// TIA Portal V16 export
// export: Created 2021-04-06T19:52:13.8560566Z, ExportSetting WithDefaults, DisplayName Totally Integrated Automation Portal, DisplayVersion V16, DisplayName TIA Portal Version Control Interface, DisplayVersion V16, DisplayName TIA Portal Openness, DisplayVersion V16, DisplayName STEP 7 Professional, DisplayVersion V16, DisplayName STEP 7 Safety, DisplayVersion V16, DisplayName WinCC Unified SCADA Engineering System, DisplayVersion V16
FUNCTION_BLOCK "ManualMode"   // FB10, LAD
{ S7_Optimized_Access := 'TRUE' }
VERSION : 0.1
// stored: AutoNumber false, IsIECCheckEnabled false, IsRetainMemResEnabled false, MemoryReserve 100, SetENOAutomatically false, UDAEnableTagReadback false
   VAR
      Bunker_Left : Array[0..12] of "controlValve";
      Bunker_Right { S7_SetPoint := 'True'} : Array[0..12] of "controlValve";
      Door { S7_SetPoint := 'True'} : Array[0..12] of "controlValve";
      flipper : "controlValve";
      runAll : Struct
         vibroLot : Bool;
      END_STRUCT;
      stopAlarm { S7_SetPoint := 'True'} : Bool;   // Стоп для блоков управления задвижками
   END_VAR
   VAR_TEMP
      i : Int;
   END_VAR
BEGIN

REGION Network 1: формирование AlarmStop
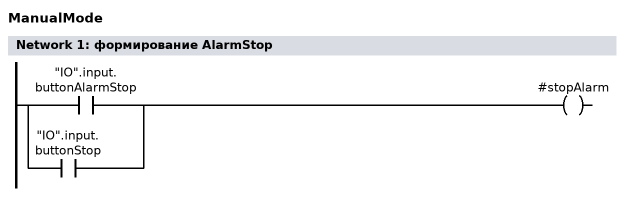
   RUNG wire#powerrail
      Contact( "IO".input.buttonAlarmStop )
      wire#w1
      Coil( #stopAlarm )
   END_RUNG
   RUNG wire#powerrail
      Contact( "IO".input.buttonStop )
   END_RUNG wire#w1
   // the same network as SCL:
   #stopAlarm := "IO".input.buttonAlarmStop OR "IO".input.buttonStop;
END_REGION

REGION Network 2 (SCL): ручное управление
   #i := 0;
   FOR #i := 1 TO 12 DO
       //если имеется разрешение на включение механизмов в ручном режиме
       IF "signalKVSStation".enableManualMode THEN
           //Bunker_left
           #Bunker_Left[#i](openQ => "signalKVSStation".qManualMode.Bunker_leftOpen[#i],
                            closeQ => "signalKVSStation".qManualMode.Bunker_leftClose[#i],
                            open := "hmi".weightLine[#i].manOpenLeftValveWeightPocket,
                            close := "hmi".weightLine[#i].manCloseLeftValveWeightPocket,
                            "time_open/close" := t#250ms,
                            stopAlarm := #stopAlarm);


           //Bunker_right
           #Bunker_Right[#i](openQ => "signalKVSStation".qManualMode.Bunker_rightOpen[#i],
                             closeQ => "signalKVSStation".qManualMode.Bunker_rightClose[#i],
                             open := "hmi".weightLine[#i].manOpenRightValveWeightPocket,
                             close := "hmi".weightLine[#i].manCloseRightValveWieghtPocket,
                             "time_open/close" := t#250ms,
                             stopAlarm := #stopAlarm);

           //Door
           #Door[#i](openQ => "signalKVSStation".qManualMode.Door_open[#i],
                     closeQ => "signalKVSStation".qManualMode.Door_close[#i],
                     open := "hmi".weightLine[#i].manOpenValveAfterVibroLot,
                     close := "hmi".weightLine[#i].manCloseValveAfterVibroLot,
                     "time_open/close" := t#250ms,
                     stopAlarm := #stopAlarm);

           //vibroLot
           IF "hmi".weightLine[#i].manVibroLotStart THEN
               "signalKVSStation".qManualMode.vibroLot[#i] := true;
           ELSE
               "signalKVSStation".qManualMode.vibroLot[#i] := false;
           END_IF;

           //теперь все что на два цикла
           IF #i = 1 OR #i = 2 THEN

               //Conv_FRV //Conv_REV
               IF "hmi".outConvAndPack[#i].manStartOutConv THEN
                   IF "hmi".outConvAndPack[#i].manIsUpConv THEN
                       "signalKVSStation".qManualMode.Conv_FRV[#i] := true;
                       "signalKVSStation".qManualMode.Conv_REV[#i] := false;
                   ELSE
                       "signalKVSStation".qManualMode.Conv_REV[#i] := true;
                       "signalKVSStation".qManualMode.Conv_FRV[#i] := false;
                   END_IF;
               ELSE
                   "signalKVSStation".qManualMode.Conv_REV[#i] := false;
                   "signalKVSStation".qManualMode.Conv_FRV[#i] := false;
               END_IF;


               //vibroTable
               IF "hmi".addedVibro.manStartVibroTable[#i] THEN
                   "signalKVSStation".qManualMode.vibroTable[#i] := true;
               ELSE
                   "signalKVSStation".qManualMode.vibroTable[#i] := false;
               END_IF;


           END_IF;

           // //flipper
           #flipper(openQ => "signalKVSStation".qManualMode.flipper_Up,
                    closeQ => "signalKVSStation".qManualMode.flipper_Down,
                    open := "hmi".plavnik.manOpenPlavnik,
                    close := "hmi".plavnik.manClosePlavnik,
                    "time_open/close" := t#250ms,
                    stopAlarm := #stopAlarm);
           //питатель
           IF "hmi".sourceConv.manStartConv THEN
               "signalKVSStation".qManualMode.startInConv := true;
           ELSE
               "signalKVSStation".qManualMode.startInConv := false;
           END_IF;

       ELSE
           //деактивируем сигналы на катушки ручного режима и
           //сигналы управления в ручном режиме
           "hmi".weightLine[#i].manOpenLeftValveWeightPocket := false;
           "signalKVSStation".qManualMode.Bunker_leftOpen[#i] := false;

           "hmi".weightLine[#i].manCloseLeftValveWeightPocket := false;
           "signalKVSStation".qManualMode.Bunker_leftClose[#i] := false;

           "hmi".weightLine[#i].manOpenRightValveWeightPocket := false;
           "signalKVSStation".qManualMode.Bunker_rightOpen[#i] := false;

           "hmi".weightLine[#i].manCloseRightValveWieghtPocket := false;
           "signalKVSStation".qManualMode.Bunker_rightClose[#i] := false;

           "hmi".weightLine[#i].manOpenRightValveWeightPocket := false;
           "signalKVSStation".qManualMode.Door_open[#i] := false;

           "hmi".weightLine[#i].manCloseValveAfterVibroLot := false;
           "signalKVSStation".qManualMode.Door_close[#i] := false;

           "hmi".weightLine[#i].manVibroLotStart := false;
           "signalKVSStation".qManualMode.vibroLot[#i] := false;
           IF #i = 1 OR #i = 2 THEN
               "hmi".outConvAndPack[#i].manStartOutConv := false;
               "signalKVSStation".qManualMode.Conv_FRV[#i] := false;
               "signalKVSStation".qManualMode.Conv_REV[#i] := false;

               "hmi".addedVibro.manStartVibroTable[#i] := false;
               "signalKVSStation".qManualMode.vibroTable[#i] := false;
           END_IF;
           "hmi".plavnik.manOpenPlavnik := false;
           "signalKVSStation".qManualMode.flipper_Up := false;

           "hmi".plavnik.manClosePlavnik := false;
           "signalKVSStation".qManualMode.flipper_Down := false;

           "hmi".sourceConv.manStartConv := false;
           "signalKVSStation".qManualMode.startInConv := false;



       END_IF;
   END_FOR;
END_REGION

REGION Network 3 (SCL): Части программы которые запускают сразу все однотипные узлы
   //запустить и остановить все вибролотки
   //
   #i := 0;
   FOR #i := 1 TO 12 DO
       IF "hmi".manRunAllVibroLot THEN
           "hmi".weightLine[#i].manVibroLotStart := true;
       END_IF;
       IF "hmi".manStopAllVibroLot THEN
           "hmi".weightLine[#i].manVibroLotStart := false;
       END_IF;
   END_FOR;
END_REGION
END_FUNCTION_BLOCK
